{attribute 'qualified_only'}
{attribute 'strict'}
TYPE Sensors :
(
	Sick,
	Pilz,
	Parker,
	Bosch
);
END_TYPE

(* stored: Version 1.1.0.1, ProductVersion 3.1.4024.12
   DUT Sensors: Id {a45ddb2d-5070-4d3b-ad16-e865ae01f7bc} *)
